// TIA Portal V21 export
FUNCTION_BLOCK "AnalogOutputScaling"   // FB11, LAD
{ S7_Optimized_Access := 'FALSE' }
// stored: SetENOAutomatically false
   VAR_INPUT
      AlwaysTrue : Bool;
      AlwaysFalse : Bool;
      MinOperatingRpm : Real;
      MaxOperatingRpm : Real;
      MaxRpm : Real;
      ManualRpm : Real;
      ActualRpm : Real;
   END_VAR
   VAR_OUTPUT
      Output : Int;
   END_VAR
   VAR
      Temp : Real;
   END_VAR
BEGIN

REGION Network 1: Scaling
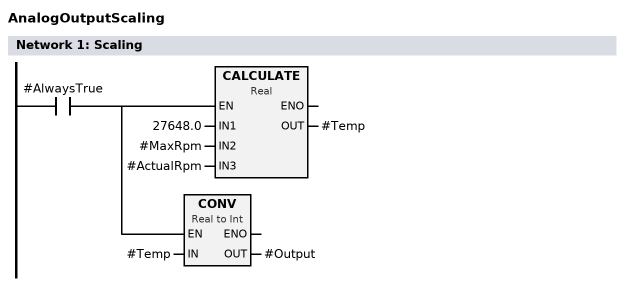
   RUNG wire#powerrail
      Contact( #AlwaysTrue )
      wire#w1
      { S7_Templates := "SrcType := Real"; S7_GenerateENO := "TRUE"; S7_Expression := "(in1*IN3)/IN2" } Calculate(in1 := 27648.0, in2 := #MaxRpm, in3 := #ActualRpm, out => #Temp)
   END_RUNG
   RUNG wire#w1
      { S7_Templates := "[SrcType := Real, DestType := Int]"; S7_GenerateENO := "TRUE" } Convert(in := #Temp, out => #Output)
   END_RUNG
   // the same network as SCL:
   IF #AlwaysTrue THEN
       #Temp := (27648.0*#ActualRpm)/#MaxRpm;
       #Output := REAL_TO_INT(#Temp);
   END_IF;
END_REGION
END_FUNCTION_BLOCK
